FUNCTION_BLOCK FB_SIM_MODBUS_COMM_JUMO EXTENDS FB_SIM_MODBUS_COMM_BASE
VAR_INPUT
END_VAR
VAR_OUTPUT
END_VAR
VAR
END_VAR

M_ActivityDo();

METHOD M_GetSimReply : STRING(255)
VAR_INPUT
	{attribute 'OPC.UA.DA' := '0'}
	cmd:	STRING(16);		// MODBUS command. Only first 8 bytes are used
END_VAR
VAR
	sReply:	STRING(255);
	sTmp:	STRING(8);
	i,j:	INT;
	pByte:	POINTER TO BYTE;
	rReal:	REAL;
	nRegister:	INT;
	nWords:	INT;	
END_VAR
// TODO User: Implement simulator replies in FBs that EXTEND FB_SIM_MODBUS_COMM_BASE.
//            Only case where cmd[1] = E_MODBUS_CMD_TYPE.READ should be implemented.

IF cmd[1] = E_MODBUS_CMD_TYPE.WRITE THEN
	M_GetSimReply := cmd;	// Reply is the same as the command
ELSE
	// Get register number - cmd[2..3] swapped bytes
	nRegister	:= M_ByteSwapINT(ADR(cmd[2]));

	// Get number of words - cmd[4..5] swapped bytes
	nWords	:= M_ByteSwapINT(ADR(cmd[4]));

	sReply[0]	:= cmd[0];
	sReply[1]	:= cmd[1];
	sReply[2]	:= INT_TO_BYTE(nWords * 2);
	
	IF nRegister = 16#00A4 THEN		// common data
		FOR i := 1 TO 54 DO
			sTmp := M_ByteSwap_REAL_TO_STRING(M_GenerateRandom_REAL(100.0,10));
			FOR j := 0 TO 3 DO
				sReply[3 + (i-1)*4 + j]	:= sTmp[j];
			END_FOR
		END_FOR
		// - Switch Stats, offset 3 + 54x4 = 219 (111 is not correct!!!)
		FOR i := 1 TO 8 DO
			sTmp := M_ByteSwap_INT_TO_STRING(M_GenerateRandom_INT(0.5,1.0));
			FOR j := 0 TO 1 DO
				sReply[111 + (i-1)*2 + j]	:= sTmp[j];
			END_FOR
		END_FOR
	ELSIF nRegister = 16#083C THEN	// set points
		FOR i := 1 TO 16 DO
			sTmp := M_ByteSwap_REAL_TO_STRING(M_GenerateRandom_REAL(80.0,1.0));
			FOR j := 0 TO 3 DO
				sReply[3 + (i-1)*4 + j]	:= sTmp[j];
			END_FOR
		END_FOR
	END_IF
	
	// TODO
	// Calculate CRC for the first 6 bytes
	//	crc	:= M_CRC(ADR(cmd),6);
	

	M_GetSimReply := sReply;
END_IF
END_METHOD

END_FUNCTION_BLOCK

(* stored: Version 1.1.0.1, ProductVersion 3.1.4024.3
   POU FB_SIM_MODBUS_COMM_JUMO: Id {e00d1754-80cf-4ee4-b64d-13d42ce8724c}, SpecialFunc None
   Method M_GetSimReply: Id {d55cb1d1-ab16-4047-bf4e-dd249b10e8d6} *)
